PROGRAM MAIN
VAR
END_VAR

P_BacnetRev14();

END_PROGRAM

(* stored: Version 1.1.0.1, ProductVersion 3.1.4024.0
   POU MAIN: Id {68ca3259-c507-4a51-90ed-2f1409c5a1ce}, SpecialFunc None *)
